# EPICS autosave request: iocBoot/generic_motors_ioc/dbSave/auto_settings.req
file COL_St_.req  P=23d:
file XY_P2_.req  P=23d:
file XY_P3_.req  P=23d:
file XY_P4_.req  P=23d:
file XY_P5_.req  P=23d:
file XY_P6_.req  P=23d:
file XY_P7_.req  P=23d:
file XY_P8_.req  P=23d:
file XY_P9_.req  P=23d:
file HS_Av_.req  P=23d:
file HS_Ah_.req  P=23d:
file XY_P12_.req  P=23d:
file XY_P13_.req  P=23d:
file XY_P14_.req  P=23d:
file XY_P15_.req  P=23d:
file XY_P16_.req  P=23d:
